(* IEC 61131-3 sources: ServoControl_Assembly_testing/, 4 files *)

(* ---- GlobalVars.var ---- *)
(* ============================================================
   GLOBAL VARIABLE DECLARATIONS
   pCO5+ Large — Ammonia Suction Servo Control
   Network: pLAN  |  Author: Tantasins  |  Rev: 2.8.3
   ============================================================ *)

VAR_GLOBAL

  (* --- Analog Inputs ---------------------------------------- *)
  rPressureRaw    : REAL;   (* AI1: 4-20mA pressure sensor, bar *)
  rPressureBar    : REAL;   (* Scaled engineering value, bar     *)

  (* --- pLAN Servo Drive I/O (node address 1) ---------------- *)
  rServoPosFbk    : REAL;   (* Servo position feedback, 0.0-100.0 % *)
  rServoPosCmd    : REAL;   (* Position command to drive, 0.0-100.0 % *)
  bServoDriveFault: BOOL;   (* Drive fault bit from pLAN           *)
  bServoEnabled   : BOOL;   (* Drive enable command               *)
  bServoHomed     : BOOL;   (* Homing complete flag               *)

  (* --- Digital Inputs --------------------------------------- *)
  bEstopHW        : BOOL;   (* Hardware E-stop (NC contact)       *)
  bNH3AlarmHW     : BOOL;   (* Ammonia gas detector (NC contact)  *)
  bManualSel      : BOOL;   (* Manual/Auto selector switch        *)

  (* --- Wireless HMI variables (pLAN or Carel pCOWeb) ------- *)
  rManualPosCmdHMI: REAL;   (* Manual position setpoint from HMI  *)
  bHMI_AutoReq    : BOOL;   (* HMI request: switch to auto        *)
  bHMI_ManualReq  : BOOL;   (* HMI request: switch to manual      *)
  bHMI_Reset      : BOOL;   (* Operator alarm reset               *)

  (* --- PID Setpoints (editable from HMI) ------------------- *)
  rPressureSP     : REAL := -0.8;  (* Suction pressure setpoint, bar *)
  rPID_Kp         : REAL := 2.5;
  rPID_Ki         : REAL := 0.4;
  rPID_Kd         : REAL := 0.1;
  rPID_OutMin     : REAL := 5.0;   (* Min valve open %, prevents slam shut *)
  rPID_OutMax     : REAL := 95.0;  (* Max valve open %                     *)

  (* --- Internal state --------------------------------------- *)
  eCtrlMode       : INT  := 0;  (* 0=AUTO  1=MANUAL  2=SAFE_STOP *)
  bAlarmActive    : BOOL;
  bAlarmLatched   : BOOL;
  sAlarmMsg       : STRING(40);
  rPID_Error      : REAL;
  rPID_Integral   : REAL;
  rPID_PrevError  : REAL;
  rPID_Output     : REAL;
  tScanTime       : TIME  := T#500MS;   (* PID scan cycle  *)

END_VAR

(* ---- FC_PID_Control.st ---- *)
(* ============================================================
   FUNCTION: Discrete PID Controller
   Positional form with anti-windup and output clamping
   ============================================================ *)

FUNCTION FC_PID_Control : VOID

  VAR_TEMP
    rDt         : REAL;
    rDerivative : REAL;
    rRawOutput  : REAL;
  END_VAR

  rDt := TIME_TO_REAL(tScanTime) / 1000.0;   (* seconds *)

  (* Error = setpoint - process variable *)
  rPID_Error := rPressureSP - rPressureBar;

  (* Integral with anti-windup clamp *)
  rPID_Integral := rPID_Integral + (rPID_Ki * rPID_Error * rDt);
  rPID_Integral := LIMIT(rPID_OutMin, rPID_Integral, rPID_OutMax);

  (* Derivative on measurement (avoids derivative kick on SP change) *)
  rDerivative := rPID_Kd * (rPID_Error - rPID_PrevError) / rDt;

  (* PID sum *)
  rRawOutput := (rPID_Kp * rPID_Error) + rPID_Integral + rDerivative;

  (* Clamp output to valve limits *)
  rPID_Output := LIMIT(rPID_OutMin, rRawOutput, rPID_OutMax);

  (* Store previous error for next scan *)
  rPID_PrevError := rPID_Error;

END_FUNCTION

(* ---- FC_WritePLAN_Servo.st ---- *)
(* ============================================================
   FUNCTION: Write servo position command via pLAN
   Uses Carel pLAN shared variable table.
   Servo drive must be configured as pLAN slave, address 1.
   Map rServoPosCmd -> pLAN shared var index 1 (REAL, 0-100%)
   Map bServoEnabled -> pLAN shared var index 2 (BOOL)
   ============================================================ *)

FUNCTION FC_WritePLAN_Servo : VOID

  (* pCOSystem pLAN write — use built-in PLAN_WRITE blocks     *)
  (* In pCO Studio: drag "pLAN Write Real" FB from library      *)
  (* and connect rServoPosCmd to it targeting node 1, var 1     *)

  (* Pseudocode representation — replace with pCO Studio FBs:  *)

  (*
    PLAN_WriteReal(
      NodeAddr  := 1,
      VarIndex  := 1,
      Value     := rServoPosCmd,
      Execute   := TRUE
    );

    PLAN_WriteBool(
      NodeAddr  := 1,
      VarIndex  := 2,
      Value     := bServoEnabled,
      Execute   := TRUE
    );

    PLAN_ReadReal(
      NodeAddr  := 1,
      VarIndex  := 3,
      Value     => rServoPosFbk,
      Execute   := TRUE
    );

    PLAN_ReadBool(
      NodeAddr  := 1,
      VarIndex  := 4,
      Value     => bServoDriveFault,
      Execute   := TRUE
    );
  *)

  (* Watchdog: if no pLAN response within 3 scans, raise fault *)
  IF NOT bServoHomed THEN
    sAlarmMsg    := 'SERVO NOT HOMED';
    bAlarmActive := TRUE;
  END_IF;

END_FUNCTION

(* ---- MainProgram.st ---- *)
(* ============================================================
   MAIN PROGRAM — Ammonia Suction Servo Control
   pCO5+ Large | pCOSystem IDE | IEC 61131-3 Structured Text
   Scan cycle: 500 ms "**IMPORTANT Testing**"
   ============================================================ *)

PROGRAM MainControl

  (* ---------------------------------------------------------- *)
  (* STEP 1: Read & scale pressure sensor                       *)
  (*   AI1 range: 4-20mA mapped to 0.0-100.0 raw units by pCO  *)
  (*   Sensor range: -1.6 bar to +0.0 bar (typical NH3 suction) *)
  (* ---------------------------------------------------------- *)
  rPressureBar := (rPressureRaw / 100.0) * 1.6 - 1.6;
  (* Result: -1.6 bar (raw=0) to 0.0 bar (raw=100) *)

  (* ---------------------------------------------------------- *)
  (* STEP 2: Safety interlock evaluation                        *)
  (*   bEstopHW and bNH3AlarmHW are NORMALLY CLOSED contacts.   *)
  (*   A TRUE signal here means the contact OPENED = danger.    *)
  (* ---------------------------------------------------------- *)
  IF bEstopHW OR bNH3AlarmHW OR bServoDriveFault THEN
    eCtrlMode    := 2;       (* Force SAFE_STOP mode *)
    bAlarmActive := TRUE;
    bAlarmLatched := TRUE;
    IF bEstopHW THEN
      sAlarmMsg := 'E-STOP ACTIVATED';
    ELSIF bNH3AlarmHW THEN
      sAlarmMsg := 'NH3 GAS ALARM - EVACUATE';
    ELSIF bServoDriveFault THEN
      sAlarmMsg := 'SERVO DRIVE FAULT';
    END_IF;
  END_IF;

  (* ---------------------------------------------------------- *)
  (* STEP 3: Alarm reset (only allowed in MANUAL mode)          *)
  (* ---------------------------------------------------------- *)
  IF bHMI_Reset AND (eCtrlMode = 1) THEN
    IF NOT bEstopHW AND NOT bNH3AlarmHW AND NOT bServoDriveFault THEN
      bAlarmLatched := FALSE;
      bAlarmActive  := FALSE;
      sAlarmMsg     := '';
    END_IF;
  END_IF;

  (* ---------------------------------------------------------- *)
  (* STEP 4: Mode switching (only when no latched alarm)        *)
  (* ---------------------------------------------------------- *)
  IF NOT bAlarmLatched THEN
    IF bHMI_AutoReq OR (NOT bManualSel) THEN
      eCtrlMode := 0;   (* AUTO *)
    ELSIF bHMI_ManualReq OR bManualSel THEN
      eCtrlMode := 1;   (* MANUAL *)
    END_IF;
  END_IF;

  (* ---------------------------------------------------------- *)
  (* STEP 5: Execute selected control mode                      *)
  (* ---------------------------------------------------------- *)
  CASE eCtrlMode OF

    0: (* ---- AUTO MODE: PID pressure control --------------- *)
       FC_PID_Control();
       rServoPosCmd := rPID_Output;
       bServoEnabled := TRUE;

    1: (* ---- MANUAL MODE: wireless HMI setpoint ------------ *)
       rServoPosCmd := LIMIT(rPID_OutMin, rManualPosCmdHMI, rPID_OutMax);
       bServoEnabled := TRUE;
       (* Reset PID integrator to prevent wind-up on mode return *)
       rPID_Integral  := rServoPosCmd;
       rPID_PrevError := rPressureBar - rPressureSP;

    2: (* ---- SAFE STOP: close valve, disable drive --------- *)
       rServoPosCmd  := rPID_OutMin;   (* Drive to minimum/closed *)
       bServoEnabled := FALSE;

  END_CASE;

  (* ---------------------------------------------------------- *)
  (* STEP 6: Write command to servo drive via pLAN              *)
  (* ---------------------------------------------------------- *)
  FC_WritePLAN_Servo();

END_PROGRAM
